// Mitsubishi GX Works2 project: 비상버튼 추가   PLC: Q02/Q02H

PROGRAM MAIN
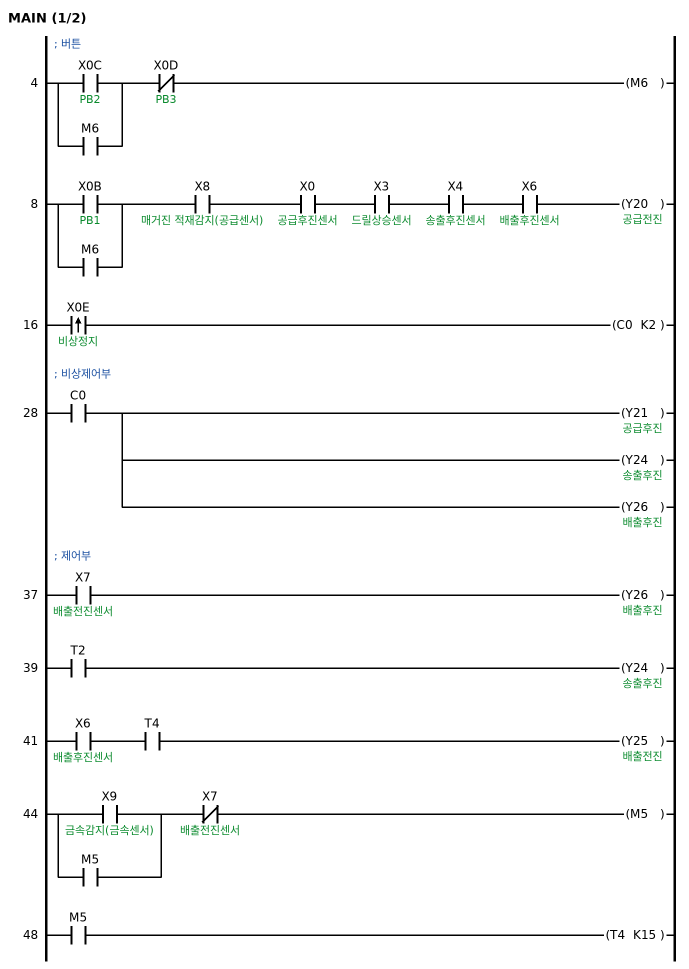
; 버튼
4     LD      X0C  ; PB2
      OR      M6
      ANI     X0D  ; PB3
      OUT     M6
8     LD      X0B  ; PB1
      OR      M6
      AND     X8  ; 매거진 적재감지(공급센서)
      AND     X0  ; 공급후진센서
      AND     X3  ; 드릴상승센서
      AND     X4  ; 송출후진센서
      AND     X6  ; 배출후진센서
      OUT     Y20  ; 공급전진
16    LDP     X0E  ; 비상정지
      OUT     C0 K2
; 비상제어부
28    LD      C0
      OUT     Y21  ; 공급후진
      OUT     Y24  ; 송출후진
      OUT     Y26  ; 배출후진
; 제어부
37    LD      X7  ; 배출전진센서
      OUT     Y26  ; 배출후진
39    LD      T2
      OUT     Y24  ; 송출후진
41    LD      X6  ; 배출후진센서
      AND     T4
      OUT     Y25  ; 배출전진
44    LD      X9  ; 금속감지(금속센서)
      OR      M5
      ANI     X7  ; 배출전진센서
      OUT     M5
48    LD      M5
      OUT     T4 K15
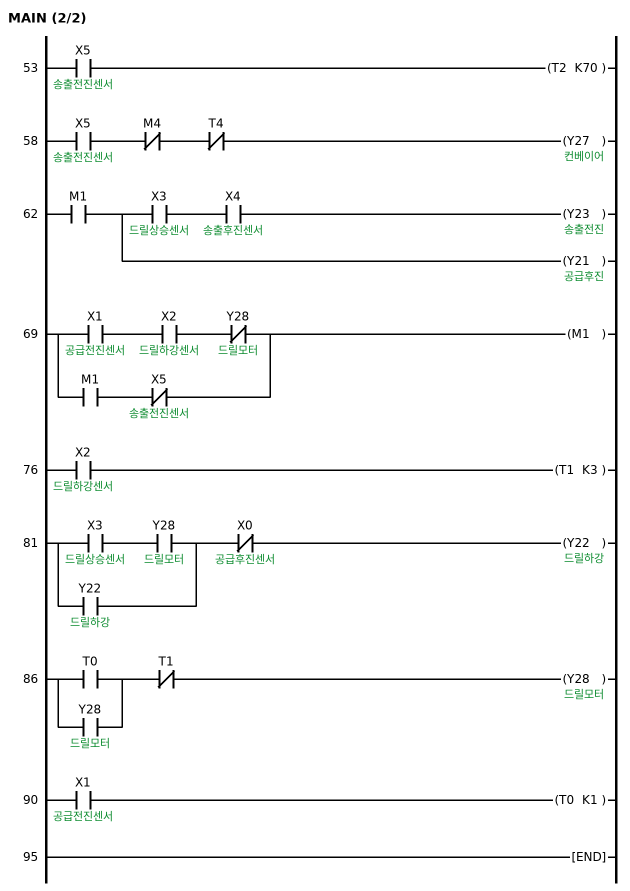
53    LD      X5  ; 송출전진센서
      OUT     T2 K70
58    LD      X5  ; 송출전진센서
      ANI     M4
      ANI     T4
      OUT     Y27  ; 컨베이어
62    LD      M1
      MPS
      AND     X3  ; 드릴상승센서
      AND     X4  ; 송출후진센서
      OUT     Y23  ; 송출전진
      MPP
      OUT     Y21  ; 공급후진
69    LD      X1  ; 공급전진센서
      AND     X2  ; 드릴하강센서
      ANI     Y28  ; 드릴모터
      LD      M1
      ANI     X5  ; 송출전진센서
      ORB
      OUT     M1
76    LD      X2  ; 드릴하강센서
      OUT     T1 K3
81    LD      X3  ; 드릴상승센서
      AND     Y28  ; 드릴모터
      OR      Y22  ; 드릴하강
      ANI     X0  ; 공급후진센서
      OUT     Y22  ; 드릴하강
86    LD      T0
      OR      Y28  ; 드릴모터
      ANI     T1
      OUT     Y28  ; 드릴모터
90    LD      X1  ; 공급전진센서
      OUT     T0 K1
95    END
END_PROGRAM

// device comments not shown above
X0A  ; 비금속 감지(가공센서)
Y29  ; 적색램프
Y2A  ; 황색램프
Y2B  ; 녹색램프
